DATA_BLOCK "DBTI"
{ S7_Optimized_Access := 'TRUE' }
VERSION : 0.1
NON_RETAIN
   VAR
      TI : Array[0..10] of "TI";
   END_VAR


BEGIN

END_DATA_BLOCK
